(* Logix 5000 project; controller AB_DataAcquisition 1769-L16ER-BB1B rev 32.11; software revision 32.02 *)

TASK MainTask (continuous, watchdog 500 ms) : MainProgram

MODULES
   Local : 1769-L16ER-BB1B (PointIO 0, rev 32.11)
      Discrete_IO : Embedded (PointIO 1, rev 32.11, Output RPI 20 ms)
END_MODULES

VAR_GLOBAL   (* controller tags *)
   LogixData1 : REAL := 1.1;
   LogixData2 : REAL := 2.2;
   LogixData3 : REAL := 3.3;
   LogixData4 : REAL := 4.4;
   LogixData5 : REAL := 5.5;
   LogixDataUnit1 : STRING := 'N';
   LogixDataUnit2 : STRING := 'Lbs';
   LogixDataUnit3 : STRING := 'Ft';
   LogixDataUnit4 : STRING := 'In';
   LogixDataUnit5 : STRING := 'Meters';
END_VAR

PROGRAM MainProgram   (* main routine MainRoutine *)

ROUTINE MainRoutine   (* ladder *)
END_ROUTINE
END_PROGRAM
